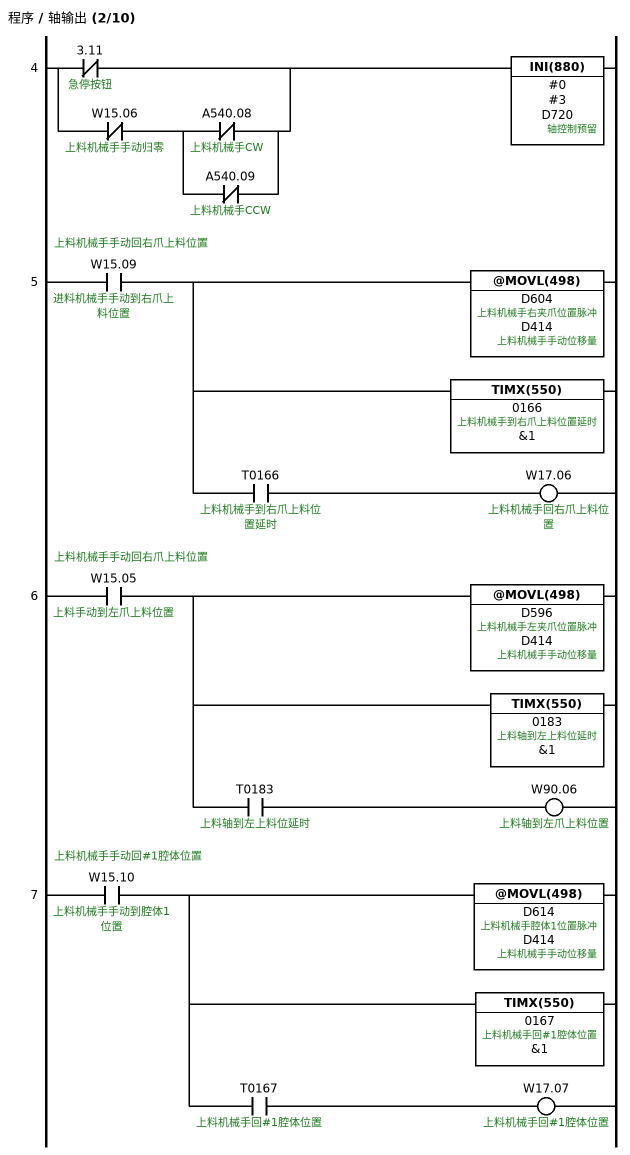
; [picture p144: 程序 / 轴输出, rungs 4-7]
; rung 4
LDNOT 3.11  ; 急停按钮
LDNOT W15.06  ; 上料机械手手动归零
LDNOT A540.08  ; 上料机械手CW
ORNOT A540.09  ; 上料机械手CCW
ANDLD
ORLD
INI(880) #0 #3 D720  ; 轴控制预留
; rung 5: 上料机械手手动回右爪上料位置
LD W15.09  ; 进料机械手手动到右爪上料位置
@MOVL(498) D604 D414  ; 上料机械手右夹爪位置脉冲, 上料机械手手动位移量
TIMX(550) 0166 &1  ; 上料机械手到右爪上料位置延时
AND T0166  ; 上料机械手到右爪上料位置延时
OUT W17.06  ; 上料机械手回右爪上料位置
; rung 6: 上料机械手手动回右爪上料位置
LD W15.05  ; 上料手动到左爪上料位置
@MOVL(498) D596 D414  ; 上料机械手左夹爪位置脉冲, 上料机械手手动位移量
TIMX(550) 0183 &1  ; 上料轴到左上料位延时
AND T0183  ; 上料轴到左上料位延时
OUT W90.06  ; 上料轴到左爪上料位置
; rung 7: 上料机械手手动回#1腔体位置
LD W15.10  ; 上料机械手手动到腔体1位置
@MOVL(498) D614 D414  ; 上料机械手腔体1位置脉冲, 上料机械手手动位移量
TIMX(550) 0167 &1  ; 上料机械手回#1腔体位置
AND T0167  ; 上料机械手回#1腔体位置
OUT W17.07  ; 上料机械手回#1腔体位置

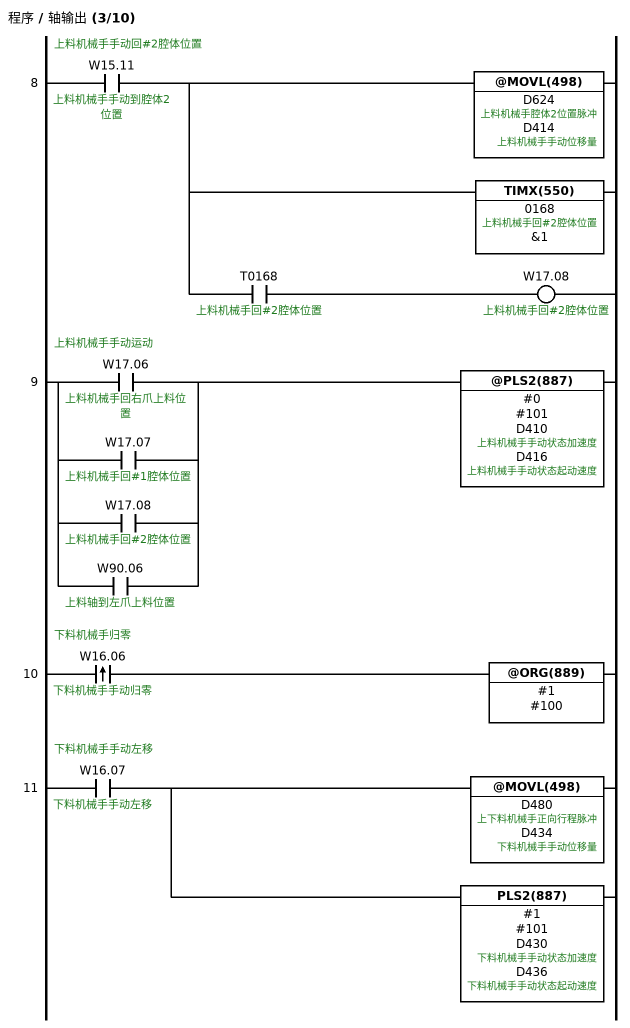
; rung 8: 上料机械手手动回#2腔体位置
LD W15.11  ; 上料机械手手动到腔体2位置
@MOVL(498) D624 D414  ; 上料机械手腔体2位置脉冲, 上料机械手手动位移量
TIMX(550) 0168 &1  ; 上料机械手回#2腔体位置
AND T0168  ; 上料机械手回#2腔体位置
OUT W17.08  ; 上料机械手回#2腔体位置
; rung 9: 上料机械手手动运动
LD W17.06  ; 上料机械手回右爪上料位置
OR W17.07  ; 上料机械手回#1腔体位置
OR W17.08  ; 上料机械手回#2腔体位置
OR W90.06  ; 上料轴到左爪上料位置
@PLS2(887) #0 #101 D410 D416  ; 上料机械手手动状态加速度, 上料机械手手动状态起动速度
; rung 10: 下料机械手归零
@LD W16.06  ; 下料机械手手动归零
@ORG(889) #1 #100
; rung 11: 下料机械手手动左移
LD W16.07  ; 下料机械手手动左移
@MOVL(498) D480 D434  ; 上下料机械手正向行程脉冲, 下料机械手手动位移量
PLS2(887) #1 #101 D430 D436  ; 下料机械手手动状态加速度, 下料机械手手动状态起动速度

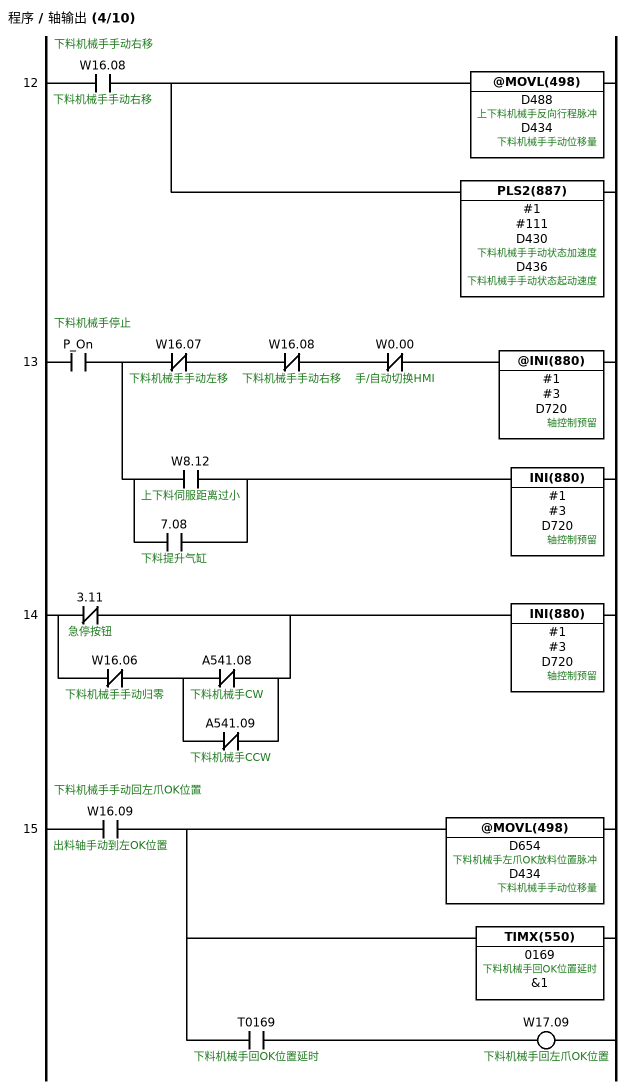
; rung 12: 下料机械手手动右移
LD W16.08  ; 下料机械手手动右移
@MOVL(498) D488 D434  ; 上下料机械手反向行程脉冲, 下料机械手手动位移量
PLS2(887) #1 #111 D430 D436  ; 下料机械手手动状态加速度, 下料机械手手动状态起动速度
; rung 13: 下料机械手停止
LD P_On
OUT TR0
ANDNOT W16.07  ; 下料机械手手动左移
ANDNOT W16.08  ; 下料机械手手动右移
ANDNOT W0.00  ; 手/自动切换HMI
@INI(880) #1 #3 D720  ; 轴控制预留
LD TR0
LD W8.12  ; 上下料伺服距离过小
OR 7.08  ; 下料提升气缸
ANDLD
INI(880) #1 #3 D720  ; 轴控制预留
; rung 14
LDNOT 3.11  ; 急停按钮
LDNOT W16.06  ; 下料机械手手动归零
LDNOT A541.08  ; 下料机械手CW
ORNOT A541.09  ; 下料机械手CCW
ANDLD
ORLD
INI(880) #1 #3 D720  ; 轴控制预留
; rung 15: 下料机械手手动回左爪OK位置
LD W16.09  ; 出料轴手动到左OK位置
@MOVL(498) D654 D434  ; 下料机械手左爪OK放料位置脉冲, 下料机械手手动位移量
TIMX(550) 0169 &1  ; 下料机械手回OK位置延时
AND T0169  ; 下料机械手回OK位置延时
OUT W17.09  ; 下料机械手回左爪OK位置

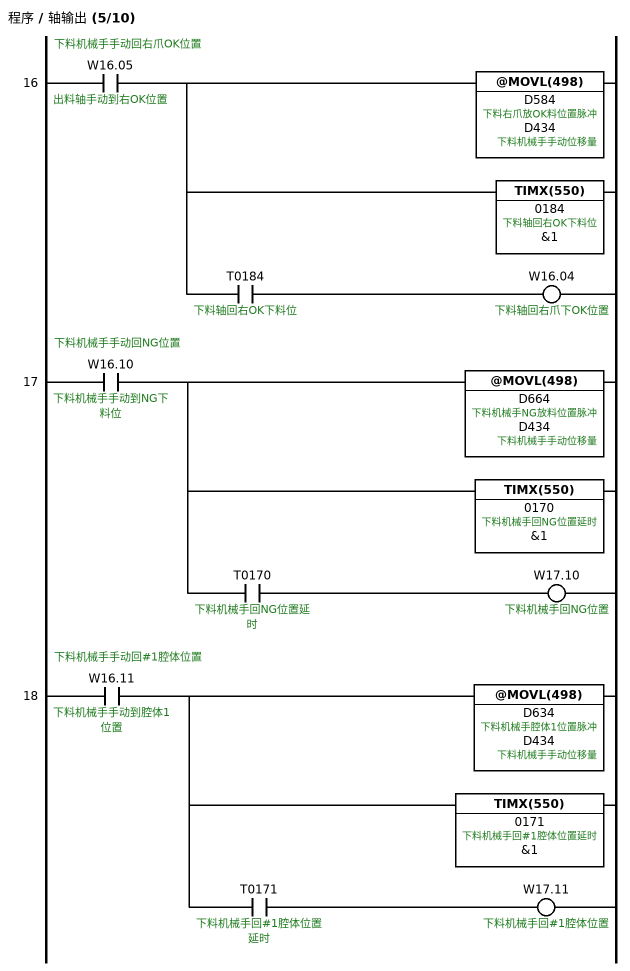
; rung 16: 下料机械手手动回右爪OK位置
LD W16.05  ; 出料轴手动到右OK位置
@MOVL(498) D584 D434  ; 下料右爪放OK料位置脉冲, 下料机械手手动位移量
TIMX(550) 0184 &1  ; 下料轴回右OK下料位
AND T0184  ; 下料轴回右OK下料位
OUT W16.04  ; 下料轴回右爪下OK位置
; rung 17: 下料机械手手动回NG位置
LD W16.10  ; 下料机械手手动到NG下料位
@MOVL(498) D664 D434  ; 下料机械手NG放料位置脉冲, 下料机械手手动位移量
TIMX(550) 0170 &1  ; 下料机械手回NG位置延时
AND T0170  ; 下料机械手回NG位置延时
OUT W17.10  ; 下料机械手回NG位置
; rung 18: 下料机械手手动回#1腔体位置
LD W16.11  ; 下料机械手手动到腔体1位置
@MOVL(498) D634 D434  ; 下料机械手腔体1位置脉冲, 下料机械手手动位移量
TIMX(550) 0171 &1  ; 下料机械手回#1腔体位置延时
AND T0171  ; 下料机械手回#1腔体位置延时
OUT W17.11  ; 下料机械手回#1腔体位置

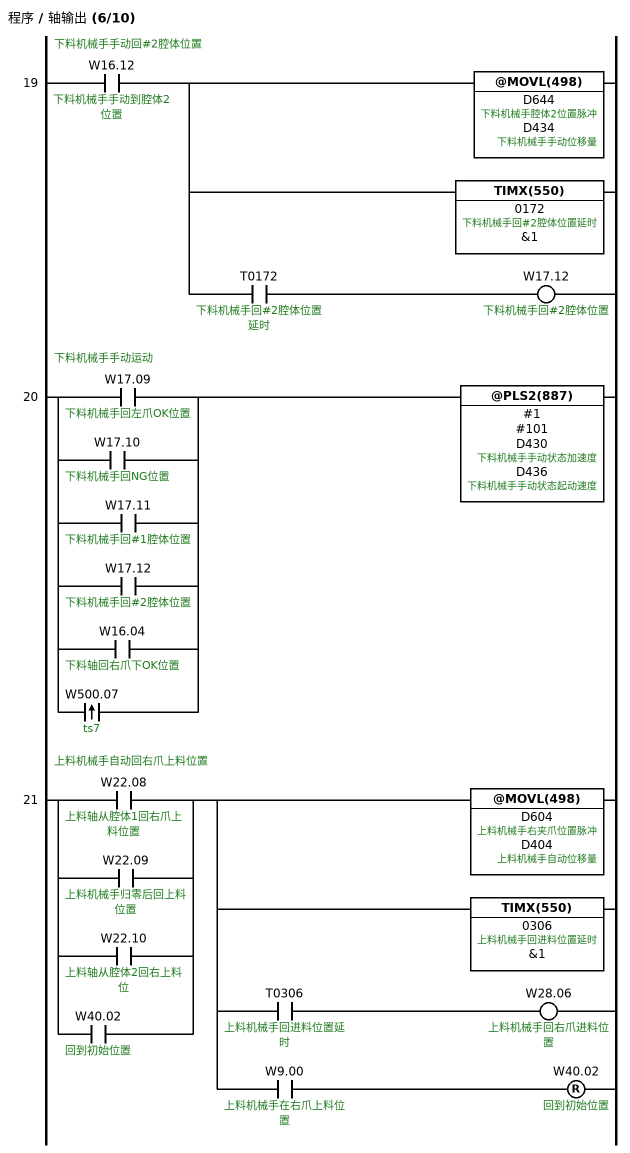
; rung 19: 下料机械手手动回#2腔体位置
LD W16.12  ; 下料机械手手动到腔体2位置
@MOVL(498) D644 D434  ; 下料机械手腔体2位置脉冲, 下料机械手手动位移量
TIMX(550) 0172 &1  ; 下料机械手回#2腔体位置延时
AND T0172  ; 下料机械手回#2腔体位置延时
OUT W17.12  ; 下料机械手回#2腔体位置
; rung 20: 下料机械手手动运动
LD W17.09  ; 下料机械手回左爪OK位置
OR W17.10  ; 下料机械手回NG位置
OR W17.11  ; 下料机械手回#1腔体位置
OR W17.12  ; 下料机械手回#2腔体位置
OR W16.04  ; 下料轴回右爪下OK位置
@OR W500.07  ; ts7
@PLS2(887) #1 #101 D430 D436  ; 下料机械手手动状态加速度, 下料机械手手动状态起动速度
; rung 21: 上料机械手自动回右爪上料位置
LD W22.08  ; 上料轴从腔体1回右爪上料位置
OR W22.09  ; 上料机械手归零后回上料位置
OR W22.10  ; 上料轴从腔体2回右上料位
OR W40.02  ; 回到初始位置
OUT TR0
@MOVL(498) D604 D404  ; 上料机械手右夹爪位置脉冲, 上料机械手自动位移量
TIMX(550) 0306 &1  ; 上料机械手回进料位置延时
AND T0306  ; 上料机械手回进料位置延时
OUT W28.06  ; 上料机械手回右爪进料位置
LD TR0
AND W9.00  ; 上料机械手在右爪上料位置
RSET W40.02  ; 回到初始位置

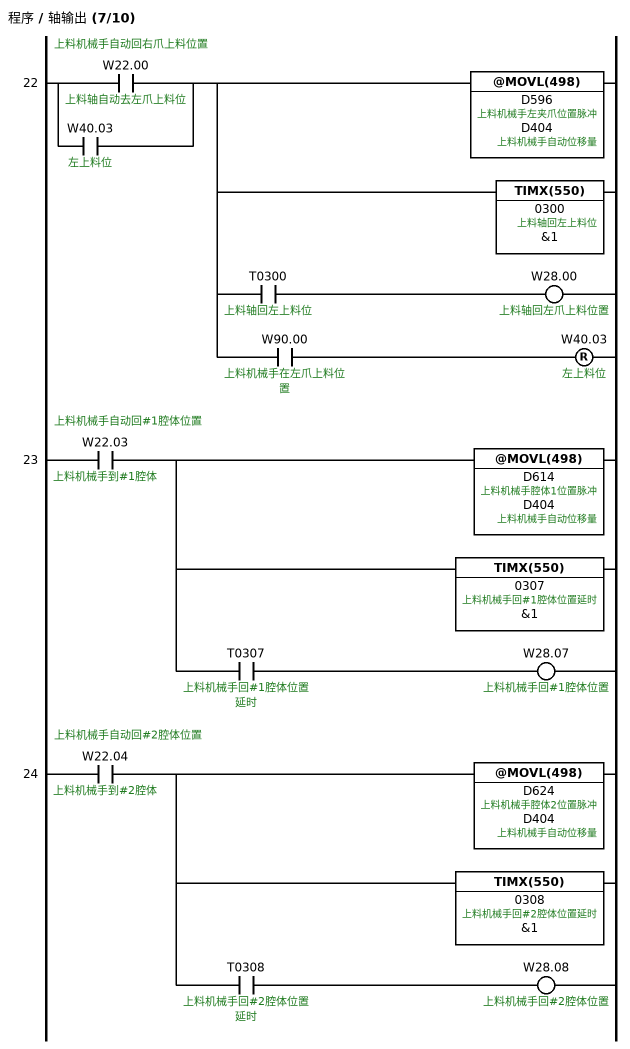
; rung 22: 上料机械手自动回右爪上料位置
LD W22.00  ; 上料轴自动去左爪上料位
OR W40.03  ; 左上料位
OUT TR0
@MOVL(498) D596 D404  ; 上料机械手左夹爪位置脉冲, 上料机械手自动位移量
TIMX(550) 0300 &1  ; 上料轴回左上料位
AND T0300  ; 上料轴回左上料位
OUT W28.00  ; 上料轴回左爪上料位置
LD TR0
AND W90.00  ; 上料机械手在左爪上料位置
RSET W40.03  ; 左上料位
; rung 23: 上料机械手自动回#1腔体位置
LD W22.03  ; 上料机械手到#1腔体
@MOVL(498) D614 D404  ; 上料机械手腔体1位置脉冲, 上料机械手自动位移量
TIMX(550) 0307 &1  ; 上料机械手回#1腔体位置延时
AND T0307  ; 上料机械手回#1腔体位置延时
OUT W28.07  ; 上料机械手回#1腔体位置
; rung 24: 上料机械手自动回#2腔体位置
LD W22.04  ; 上料机械手到#2腔体
@MOVL(498) D624 D404  ; 上料机械手腔体2位置脉冲, 上料机械手自动位移量
TIMX(550) 0308 &1  ; 上料机械手回#2腔体位置延时
AND T0308  ; 上料机械手回#2腔体位置延时
OUT W28.08  ; 上料机械手回#2腔体位置

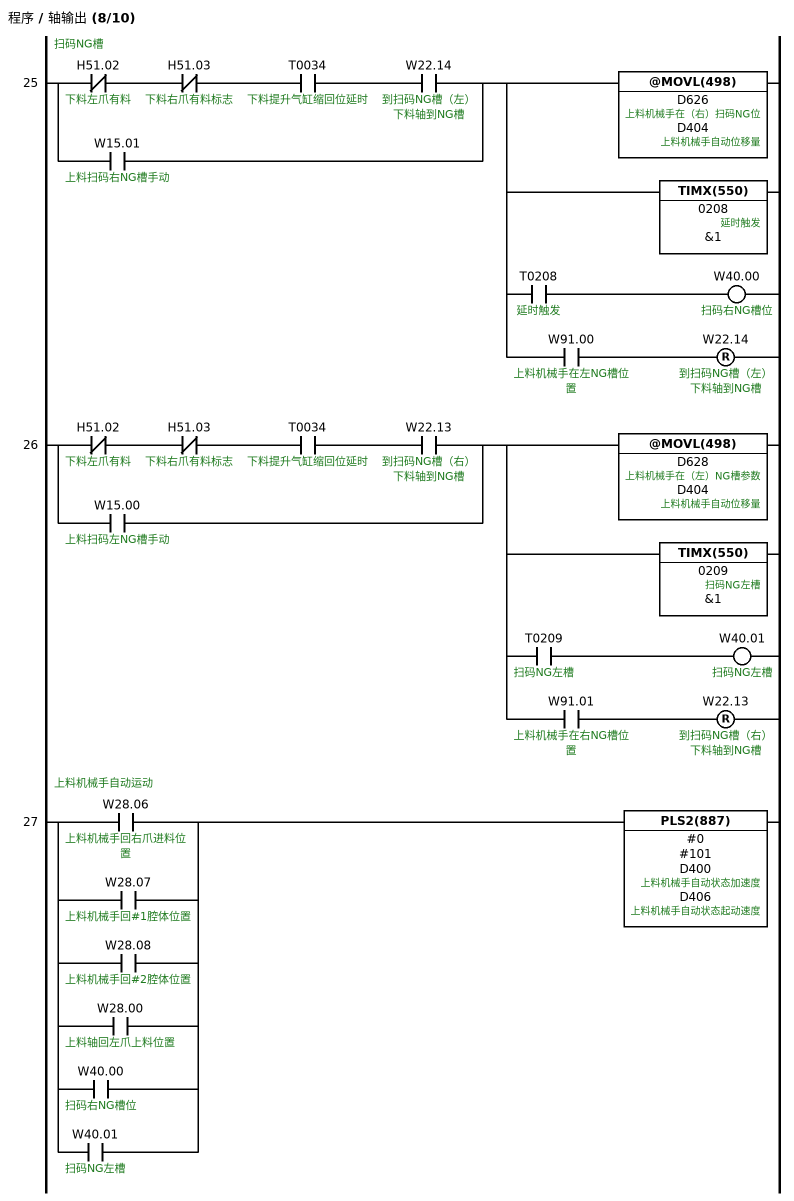
; rung 25: 扫码NG槽
LDNOT H51.02  ; 下料左爪有料
ANDNOT H51.03  ; 下料右爪有料标志
AND T0034  ; 下料提升气缸缩回位延时
AND W22.14  ; 到扫码NG槽（左） 下料轴到NG槽
OR W15.01  ; 上料扫码右NG槽手动
OUT TR0
@MOVL(498) D626 D404  ; 上料机械手在（右）扫码NG位, 上料机械手自动位移量
TIMX(550) 0208 &1  ; 延时触发
AND T0208  ; 延时触发
OUT W40.00  ; 扫码右NG槽位
LD TR0
AND W91.00  ; 上料机械手在左NG槽位置
RSET W22.14  ; 到扫码NG槽（左） 下料轴到NG槽
; rung 26
LDNOT H51.02  ; 下料左爪有料
ANDNOT H51.03  ; 下料右爪有料标志
AND T0034  ; 下料提升气缸缩回位延时
AND W22.13  ; 到扫码NG槽（右） 下料轴到NG槽
OR W15.00  ; 上料扫码左NG槽手动
OUT TR0
@MOVL(498) D628 D404  ; 上料机械手在（左）NG槽参数, 上料机械手自动位移量
TIMX(550) 0209 &1  ; 扫码NG左槽
AND T0209  ; 扫码NG左槽
OUT W40.01  ; 扫码NG左槽
LD TR0
AND W91.01  ; 上料机械手在右NG槽位置
RSET W22.13  ; 到扫码NG槽（右） 下料轴到NG槽
; rung 27: 上料机械手自动运动
LD W28.06  ; 上料机械手回右爪进料位置
OR W28.07  ; 上料机械手回#1腔体位置
OR W28.08  ; 上料机械手回#2腔体位置
OR W28.00  ; 上料轴回左爪上料位置
OR W40.00  ; 扫码右NG槽位
OR W40.01  ; 扫码NG左槽
PLS2(887) #0 #101 D400 D406  ; 上料机械手自动状态加速度, 上料机械手自动状态起动速度

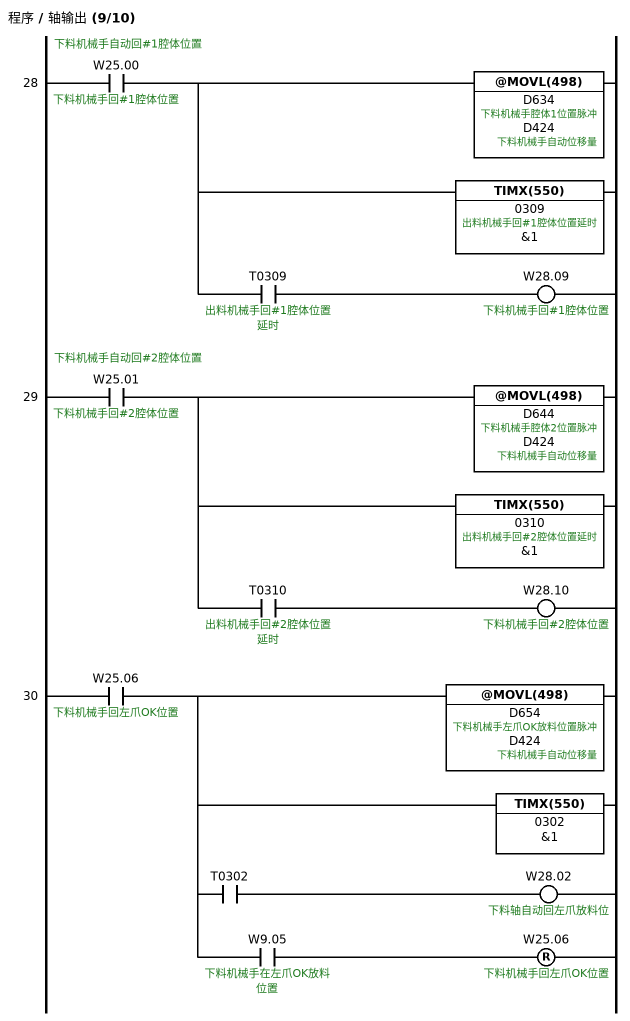
; rung 28: 下料机械手自动回#1腔体位置
LD W25.00  ; 下料机械手回#1腔体位置
@MOVL(498) D634 D424  ; 下料机械手腔体1位置脉冲, 下料机械手自动位移量
TIMX(550) 0309 &1  ; 出料机械手回#1腔体位置延时
AND T0309  ; 出料机械手回#1腔体位置延时
OUT W28.09  ; 下料机械手回#1腔体位置
; rung 29: 下料机械手自动回#2腔体位置
LD W25.01  ; 下料机械手回#2腔体位置
@MOVL(498) D644 D424  ; 下料机械手腔体2位置脉冲, 下料机械手自动位移量
TIMX(550) 0310 &1  ; 出料机械手回#2腔体位置延时
AND T0310  ; 出料机械手回#2腔体位置延时
OUT W28.10  ; 下料机械手回#2腔体位置
; rung 30
LD W25.06  ; 下料机械手回左爪OK位置
OUT TR0
@MOVL(498) D654 D424  ; 下料机械手左爪OK放料位置脉冲, 下料机械手自动位移量
TIMX(550) 0302 &1
AND T0302
OUT W28.02  ; 下料轴自动回左爪放料位
LD TR0
AND W9.05  ; 下料机械手在左爪OK放料位置
RSET W25.06  ; 下料机械手回左爪OK位置

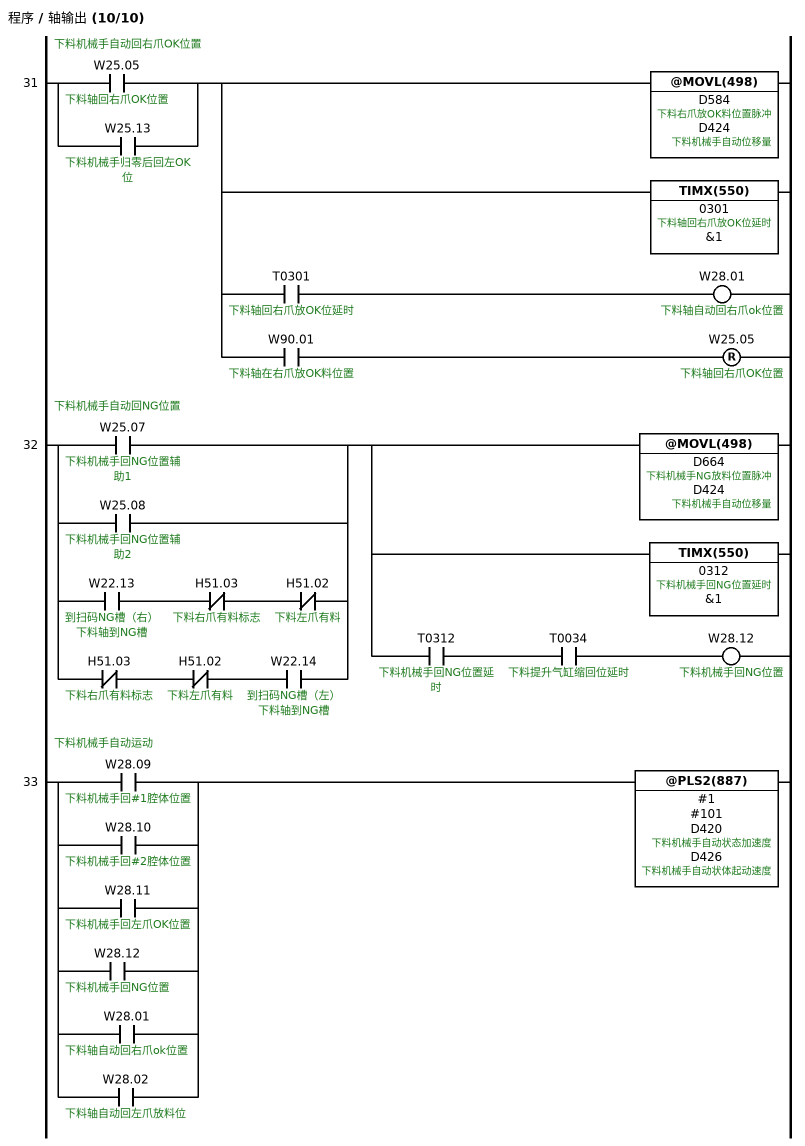
; rung 31: 下料机械手自动回右爪OK位置
LD W25.05  ; 下料轴回右爪OK位置
OR W25.13  ; 下料机械手归零后回左OK位
OUT TR0
@MOVL(498) D584 D424  ; 下料右爪放OK料位置脉冲, 下料机械手自动位移量
TIMX(550) 0301 &1  ; 下料轴回右爪放OK位延时
AND T0301  ; 下料轴回右爪放OK位延时
OUT W28.01  ; 下料轴自动回右爪ok位置
LD TR0
AND W90.01  ; 下料轴在右爪放OK料位置
RSET W25.05  ; 下料轴回右爪OK位置
; rung 32: 下料机械手自动回NG位置
LD W25.07  ; 下料机械手回NG位置辅助1
OR W25.08  ; 下料机械手回NG位置辅助2
LD W22.13  ; 到扫码NG槽（右） 下料轴到NG槽
ANDNOT H51.03  ; 下料右爪有料标志
ANDNOT H51.02  ; 下料左爪有料
ORLD
LDNOT H51.03  ; 下料右爪有料标志
ANDNOT H51.02  ; 下料左爪有料
AND W22.14  ; 到扫码NG槽（左） 下料轴到NG槽
ORLD
@MOVL(498) D664 D424  ; 下料机械手NG放料位置脉冲, 下料机械手自动位移量
TIMX(550) 0312 &1  ; 下料机械手回NG位置延时
AND T0312  ; 下料机械手回NG位置延时
AND T0034  ; 下料提升气缸缩回位延时
OUT W28.12  ; 下料机械手回NG位置
; rung 33: 下料机械手自动运动
LD W28.09  ; 下料机械手回#1腔体位置
OR W28.10  ; 下料机械手回#2腔体位置
OR W28.11  ; 下料机械手回左爪OK位置
OR W28.12  ; 下料机械手回NG位置
OR W28.01  ; 下料轴自动回右爪ok位置
OR W28.02  ; 下料轴自动回左爪放料位
@PLS2(887) #1 #101 D420 D426  ; 下料机械手自动状态加速度, 下料机械手自动状体起动速度

### Section 普通输出

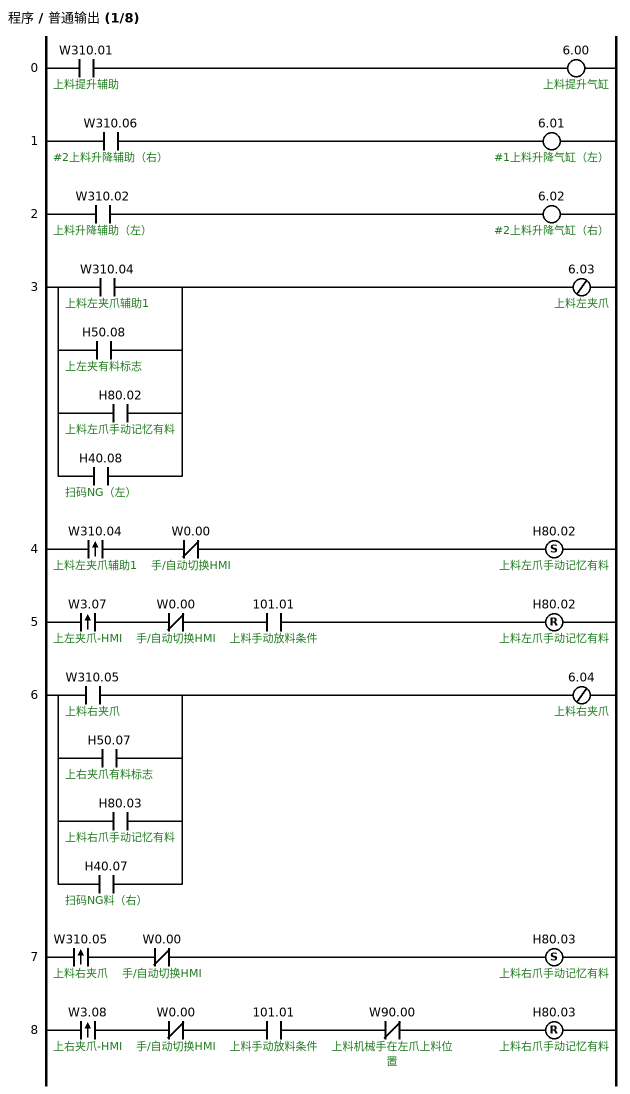
; rung 0
LD W310.01  ; 上料提升辅助
OUT 6.00  ; 上料提升气缸
; rung 1
LD W310.06  ; #2上料升降辅助（右）
OUT 6.01  ; #1上料升降气缸（左）
; rung 2
LD W310.02  ; 上料升降辅助（左）
OUT 6.02  ; #2上料升降气缸（右）
; rung 3
LD W310.04  ; 上料左夹爪辅助1
OR H50.08  ; 上左夹有料标志
OR H80.02  ; 上料左爪手动记忆有料
OR H40.08  ; 扫码NG（左）
OUTNOT 6.03  ; 上料左夹爪
; rung 4
@LD W310.04  ; 上料左夹爪辅助1
ANDNOT W0.00  ; 手/自动切换HMI
SET H80.02  ; 上料左爪手动记忆有料
; rung 5
@LD W3.07  ; 上左夹爪-HMI
ANDNOT W0.00  ; 手/自动切换HMI
AND 101.01  ; 上料手动放料条件
RSET H80.02  ; 上料左爪手动记忆有料
; rung 6
LD W310.05  ; 上料右夹爪
OR H50.07  ; 上右夹爪有料标志
OR H80.03  ; 上料右爪手动记忆有料
OR H40.07  ; 扫码NG料（右）
OUTNOT 6.04  ; 上料右夹爪
; rung 7
@LD W310.05  ; 上料右夹爪
ANDNOT W0.00  ; 手/自动切换HMI
SET H80.03  ; 上料右爪手动记忆有料
; rung 8
@LD W3.08  ; 上右夹爪-HMI
ANDNOT W0.00  ; 手/自动切换HMI
AND 101.01  ; 上料手动放料条件
ANDNOT W90.00  ; 上料机械手在左爪上料位置
RSET H80.03  ; 上料右爪手动记忆有料

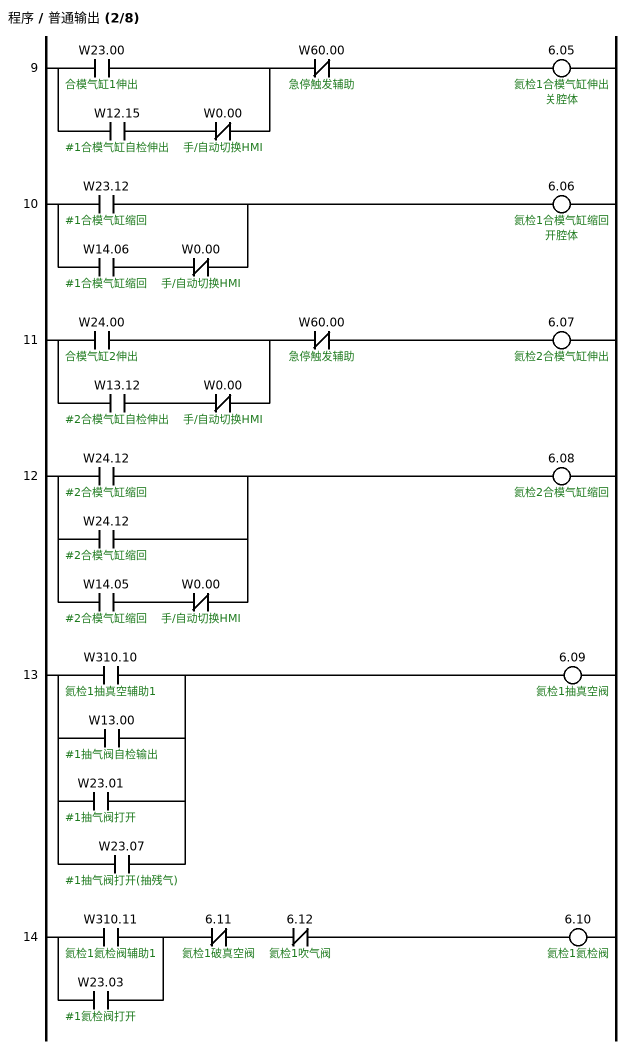
; rung 9
LD W23.00  ; 合模气缸1伸出
LD W12.15  ; #1合模气缸自检伸出
ANDNOT W0.00  ; 手/自动切换HMI
ORLD
ANDNOT W60.00  ; 急停触发辅助
OUT 6.05  ; 氦检1合模气缸伸出 关腔体
; rung 10
LD W23.12  ; #1合模气缸缩回
LD W14.06  ; #1合模气缸缩回
ANDNOT W0.00  ; 手/自动切换HMI
ORLD
OUT 6.06  ; 氦检1合模气缸缩回 开腔体
; rung 11
LD W24.00  ; 合模气缸2伸出
LD W13.12  ; #2合模气缸自检伸出
ANDNOT W0.00  ; 手/自动切换HMI
ORLD
ANDNOT W60.00  ; 急停触发辅助
OUT 6.07  ; 氦检2合模气缸伸出
; rung 12
LD W24.12  ; #2合模气缸缩回
OR W24.12  ; #2合模气缸缩回
LD W14.05  ; #2合模气缸缩回
ANDNOT W0.00  ; 手/自动切换HMI
ORLD
OUT 6.08  ; 氦检2合模气缸缩回
; rung 13
LD W310.10  ; 氦检1抽真空辅助1
OR W13.00  ; #1抽气阀自检输出
OR W23.01  ; #1抽气阀打开
OR W23.07  ; #1抽气阀打开(抽残气)
OUT 6.09  ; 氦检1抽真空阀
; rung 14
LD W310.11  ; 氦检1氦检阀辅助1
OR W23.03  ; #1氦检阀打开
ANDNOT 6.11  ; 氦检1破真空阀
ANDNOT 6.12  ; 氦检1吹气阀
OUT 6.10  ; 氦检1氦检阀

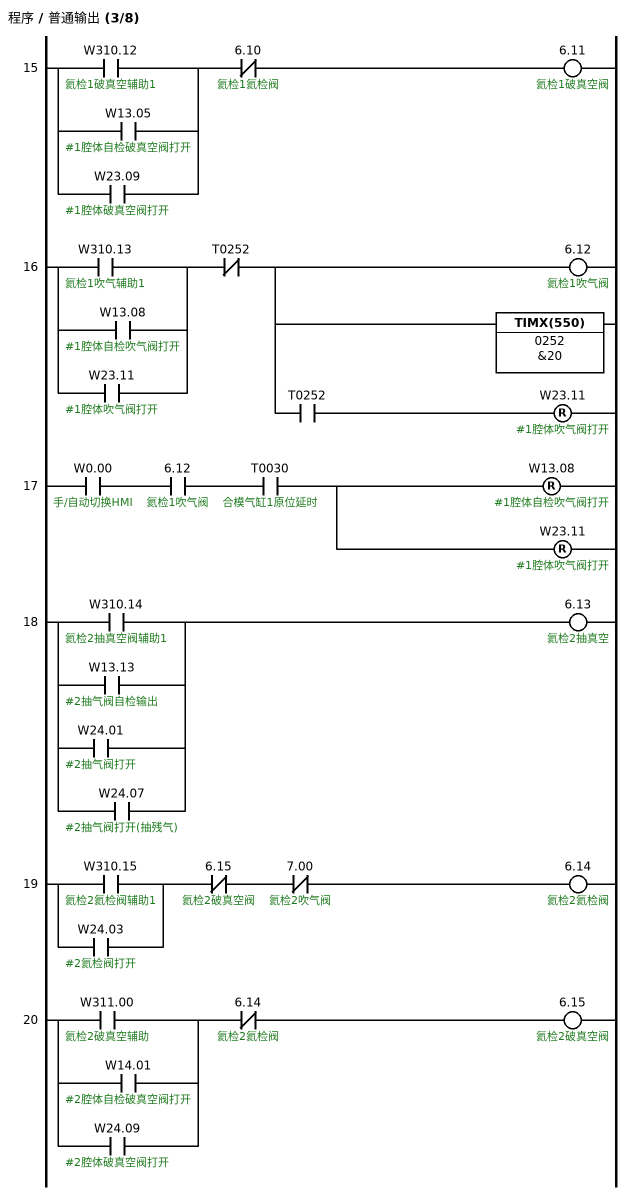
; rung 15
LD W310.12  ; 氦检1破真空辅助1
OR W13.05  ; #1腔体自检破真空阀打开
OR W23.09  ; #1腔体破真空阀打开
ANDNOT 6.10  ; 氦检1氦检阀
OUT 6.11  ; 氦检1破真空阀
; rung 16
LD W310.13  ; 氦检1吹气辅助1
OR W13.08  ; #1腔体自检吹气阀打开
OR W23.11  ; #1腔体吹气阀打开
ANDNOT T0252
OUT 6.12  ; 氦检1吹气阀
TIMX(550) 0252 &20
AND T0252
RSET W23.11  ; #1腔体吹气阀打开
; rung 17
LD W0.00  ; 手/自动切换HMI
AND 6.12  ; 氦检1吹气阀
AND T0030  ; 合模气缸1原位延时
RSET W13.08  ; #1腔体自检吹气阀打开
RSET W23.11  ; #1腔体吹气阀打开
; rung 18
LD W310.14  ; 氦检2抽真空阀辅助1
OR W13.13  ; #2抽气阀自检输出
OR W24.01  ; #2抽气阀打开
OR W24.07  ; #2抽气阀打开(抽残气)
OUT 6.13  ; 氦检2抽真空
; rung 19
LD W310.15  ; 氦检2氦检阀辅助1
OR W24.03  ; #2氦检阀打开
ANDNOT 6.15  ; 氦检2破真空阀
ANDNOT 7.00  ; 氦检2吹气阀
OUT 6.14  ; 氦检2氦检阀
; rung 20
LD W311.00  ; 氦检2破真空辅助
OR W14.01  ; #2腔体自检破真空阀打开
OR W24.09  ; #2腔体破真空阀打开
ANDNOT 6.14  ; 氦检2氦检阀
OUT 6.15  ; 氦检2破真空阀

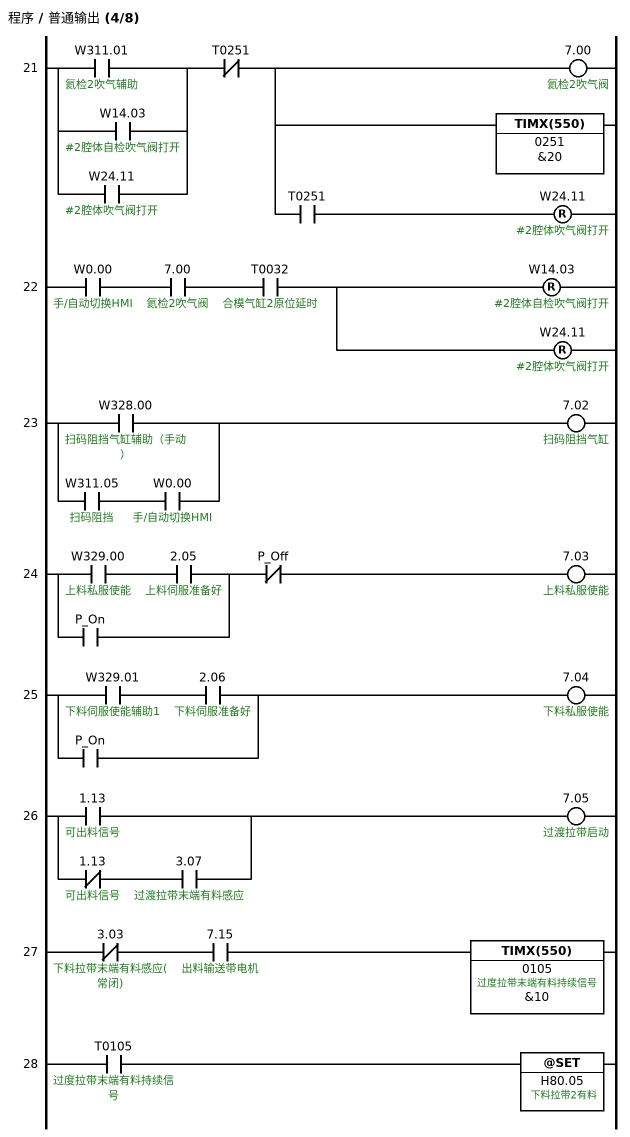
; rung 21
LD W311.01  ; 氦检2吹气辅助
OR W14.03  ; #2腔体自检吹气阀打开
OR W24.11  ; #2腔体吹气阀打开
ANDNOT T0251
OUT 7.00  ; 氦检2吹气阀
TIMX(550) 0251 &20
AND T0251
RSET W24.11  ; #2腔体吹气阀打开
; rung 22
LD W0.00  ; 手/自动切换HMI
AND 7.00  ; 氦检2吹气阀
AND T0032  ; 合模气缸2原位延时
RSET W14.03  ; #2腔体自检吹气阀打开
RSET W24.11  ; #2腔体吹气阀打开
; rung 23
LD W328.00  ; 扫码阻挡气缸辅助（手动）
LD W311.05  ; 扫码阻挡
AND W0.00  ; 手/自动切换HMI
ORLD
OUT 7.02  ; 扫码阻挡气缸
; rung 24
LD W329.00  ; 上料私服使能
AND 2.05  ; 上料伺服准备好
OR P_On
ANDNOT P_Off
OUT 7.03  ; 上料私服使能
; rung 25
LD W329.01  ; 下料伺服使能辅助1
AND 2.06  ; 下料伺服准备好
OR P_On
OUT 7.04  ; 下料私服使能
; rung 26
LD 1.13  ; 可出料信号
LDNOT 1.13  ; 可出料信号
AND 3.07  ; 过渡拉带末端有料感应
ORLD
OUT 7.05  ; 过渡拉带启动
; rung 27
LDNOT 3.03  ; 下料拉带末端有料感应(常闭)
AND 7.15  ; 出料输送带电机
TIMX(550) 0105 &10  ; 过度拉带末端有料持续信号
; rung 28
LD T0105  ; 过度拉带末端有料持续信号
@SET H80.05  ; 下料拉带2有料

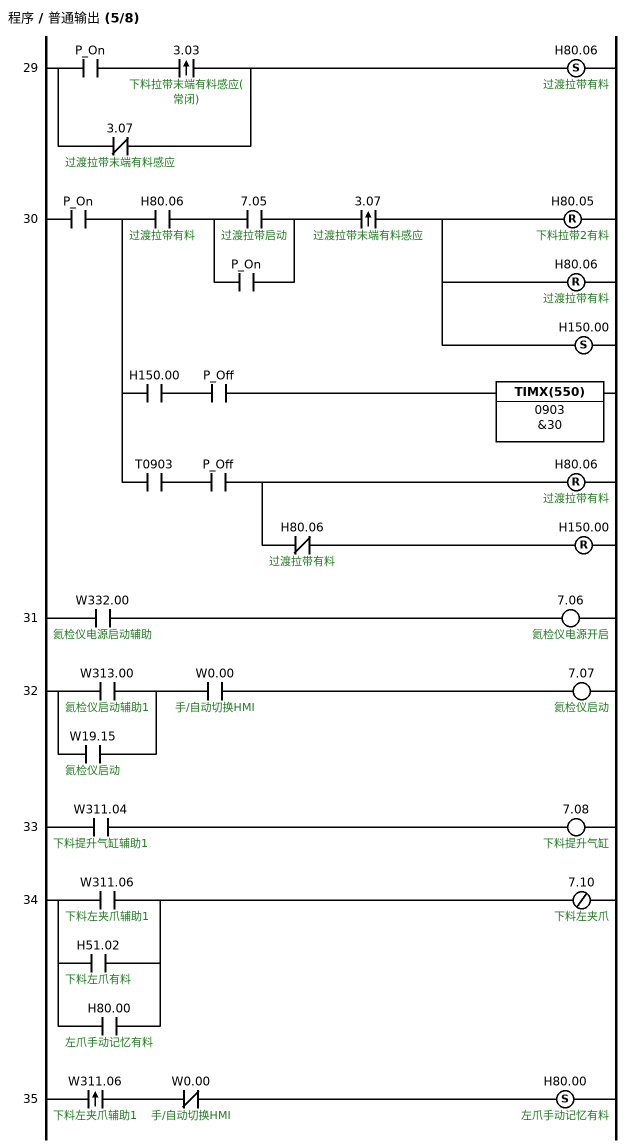
; rung 29
LD P_On
@AND 3.03  ; 下料拉带末端有料感应(常闭)
ORNOT 3.07  ; 过渡拉带末端有料感应
SET H80.06  ; 过渡拉带有料
; rung 30
LD P_On
OUT TR0
AND H80.06  ; 过渡拉带有料
LD 7.05  ; 过渡拉带启动
OR P_On
ANDLD
@AND 3.07  ; 过渡拉带末端有料感应
RSET H80.05  ; 下料拉带2有料
RSET H80.06  ; 过渡拉带有料
SET H150.00
LD TR0
AND H150.00
AND P_Off
TIMX(550) 0903 &30
LD TR0
AND T0903
AND P_Off
RSET H80.06  ; 过渡拉带有料
ANDNOT H80.06  ; 过渡拉带有料
RSET H150.00
; rung 31
LD W332.00  ; 氦检仪电源启动辅助
OUT 7.06  ; 氦检仪电源开启
; rung 32
LD W313.00  ; 氦检仪启动辅助1
OR W19.15  ; 氦检仪启动
AND W0.00  ; 手/自动切换HMI
OUT 7.07  ; 氦检仪启动
; rung 33
LD W311.04  ; 下料提升气缸辅助1
OUT 7.08  ; 下料提升气缸
; rung 34
LD W311.06  ; 下料左夹爪辅助1
OR H51.02  ; 下料左爪有料
OR H80.00  ; 左爪手动记忆有料
OUTNOT 7.10  ; 下料左夹爪
; rung 35
@LD W311.06  ; 下料左夹爪辅助1
ANDNOT W0.00  ; 手/自动切换HMI
SET H80.00  ; 左爪手动记忆有料

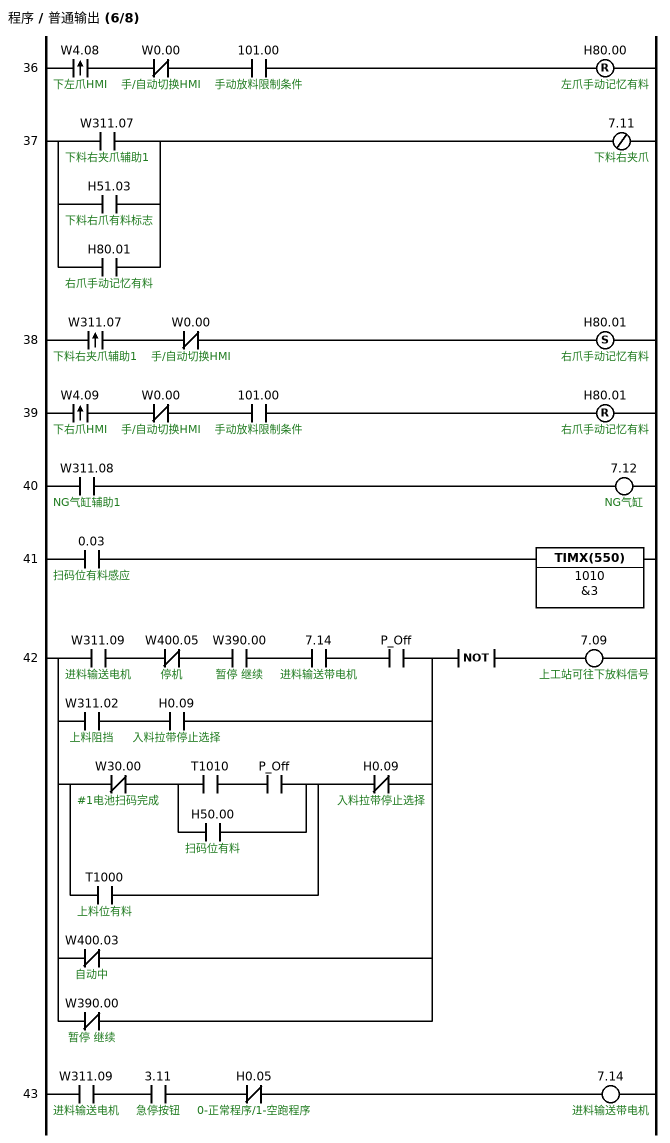
; rung 36
@LD W4.08  ; 下左爪HMI
ANDNOT W0.00  ; 手/自动切换HMI
AND 101.00  ; 手动放料限制条件
RSET H80.00  ; 左爪手动记忆有料
; rung 37
LD W311.07  ; 下料右夹爪辅助1
OR H51.03  ; 下料右爪有料标志
OR H80.01  ; 右爪手动记忆有料
OUTNOT 7.11  ; 下料右夹爪
; rung 38
@LD W311.07  ; 下料右夹爪辅助1
ANDNOT W0.00  ; 手/自动切换HMI
SET H80.01  ; 右爪手动记忆有料
; rung 39
@LD W4.09  ; 下右爪HMI
ANDNOT W0.00  ; 手/自动切换HMI
AND 101.00  ; 手动放料限制条件
RSET H80.01  ; 右爪手动记忆有料
; rung 40
LD W311.08  ; NG气缸辅助1
OUT 7.12  ; NG气缸
; rung 41
LD 0.03  ; 扫码位有料感应
TIMX(550) 1010 &3
; rung 42
LD W311.09  ; 进料输送电机
ANDNOT W400.05  ; 停机
AND W390.00  ; 暂停 继续
AND 7.14  ; 进料输送带电机
AND P_Off
LD W311.02  ; 上料阻挡
AND H0.09  ; 入料拉带停止选择
ORLD
LDNOT W30.00  ; #1电池扫码完成
LD T1010
AND P_Off
OR H50.00  ; 扫码位有料
ANDLD
OR T1000  ; 上料位有料
ANDNOT H0.09  ; 入料拉带停止选择
ORLD
ORNOT W400.03  ; 自动中
ORNOT W390.00  ; 暂停 继续
NOT(520)
OUT 7.09  ; 上工站可往下放料信号
; rung 43
LD W311.09  ; 进料输送电机
AND 3.11  ; 急停按钮
ANDNOT H0.05  ; 0-正常程序/1-空跑程序
OUT 7.14  ; 进料输送带电机

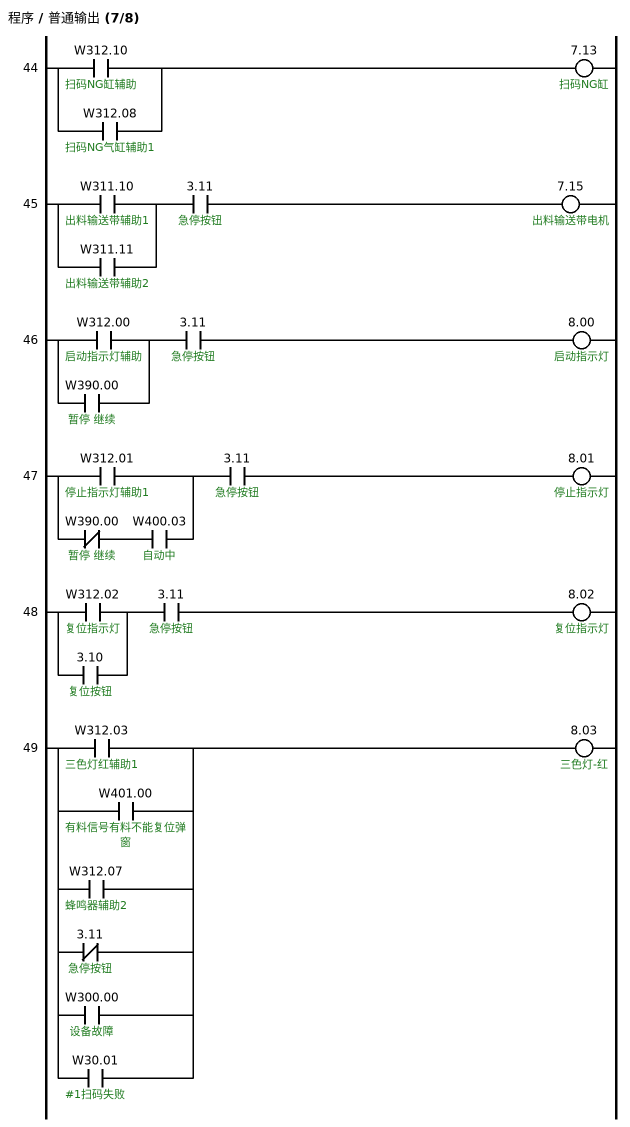
; rung 44
LD W312.10  ; 扫码NG缸辅助
OR W312.08  ; 扫码NG气缸辅助1
OUT 7.13  ; 扫码NG缸
; rung 45
LD W311.10  ; 出料输送带辅助1
OR W311.11  ; 出料输送带辅助2
AND 3.11  ; 急停按钮
OUT 7.15  ; 出料输送带电机
; rung 46
LD W312.00  ; 启动指示灯辅助
OR W390.00  ; 暂停 继续
AND 3.11  ; 急停按钮
OUT 8.00  ; 启动指示灯
; rung 47
LD W312.01  ; 停止指示灯辅助1
LDNOT W390.00  ; 暂停 继续
AND W400.03  ; 自动中
ORLD
AND 3.11  ; 急停按钮
OUT 8.01  ; 停止指示灯
; rung 48
LD W312.02  ; 复位指示灯
OR 3.10  ; 复位按钮
AND 3.11  ; 急停按钮
OUT 8.02  ; 复位指示灯
; rung 49
LD W312.03  ; 三色灯红辅助1
OR W401.00  ; 有料信号有料不能复位弹窗
OR W312.07  ; 蜂鸣器辅助2
ORNOT 3.11  ; 急停按钮
OR W300.00  ; 设备故障
OR W30.01  ; #1扫码失败
OUT 8.03  ; 三色灯-红

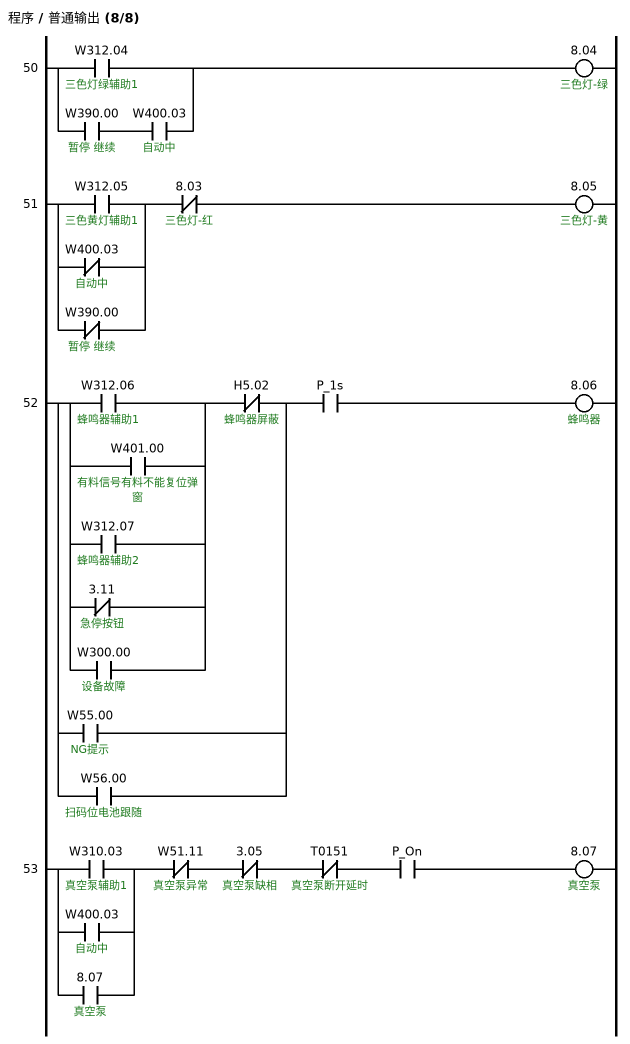
; rung 50
LD W312.04  ; 三色灯绿辅助1
LD W390.00  ; 暂停 继续
AND W400.03  ; 自动中
ORLD
OUT 8.04  ; 三色灯-绿
; rung 51
LD W312.05  ; 三色黄灯辅助1
ORNOT W400.03  ; 自动中
ORNOT W390.00  ; 暂停 继续
ANDNOT 8.03  ; 三色灯-红
OUT 8.05  ; 三色灯-黄
; rung 52
LD W312.06  ; 蜂鸣器辅助1
OR W401.00  ; 有料信号有料不能复位弹窗
OR W312.07  ; 蜂鸣器辅助2
ORNOT 3.11  ; 急停按钮
OR W300.00  ; 设备故障
ANDNOT H5.02  ; 蜂鸣器屏蔽
OR W55.00  ; NG提示
OR W56.00  ; 扫码位电池跟随
AND P_1s
OUT 8.06  ; 蜂鸣器
; rung 53
LD W310.03  ; 真空泵辅助1
OR W400.03  ; 自动中
OR 8.07  ; 真空泵
ANDNOT W51.11  ; 真空泵异常
ANDNOT 3.05  ; 真空泵缺相
ANDNOT T0151  ; 真空泵断开延时
AND P_On
OUT 8.07  ; 真空泵

### Section 氦检仪读值

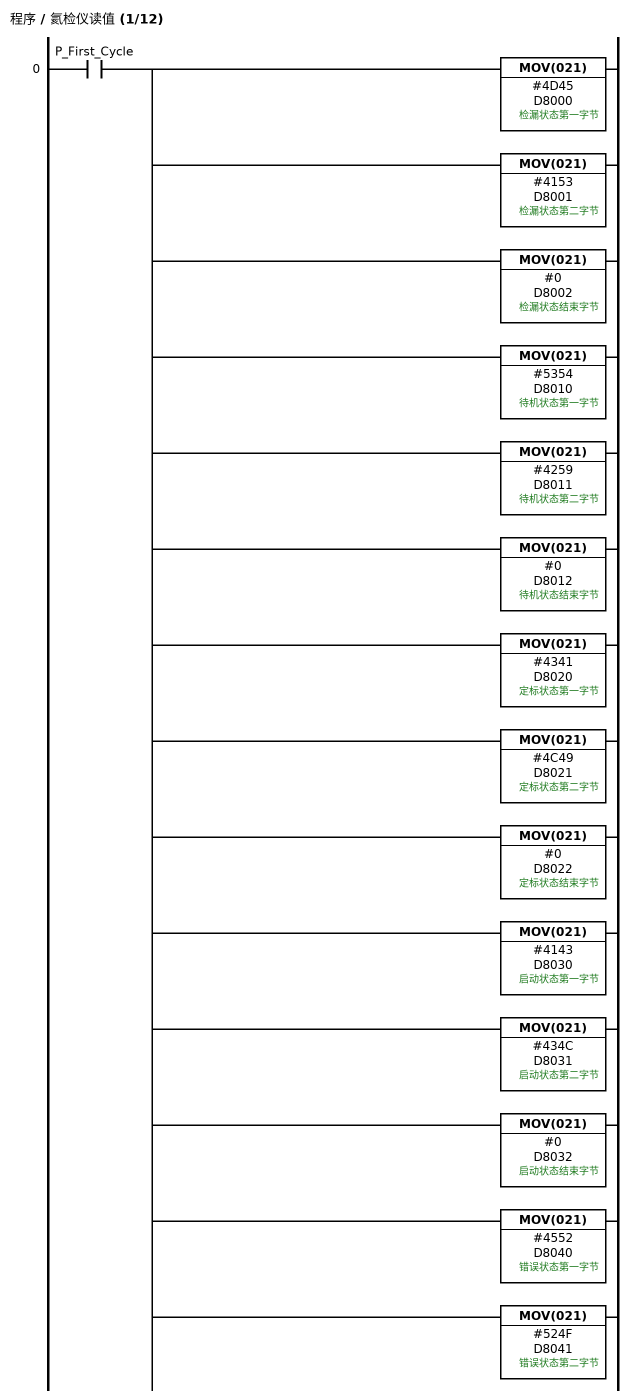

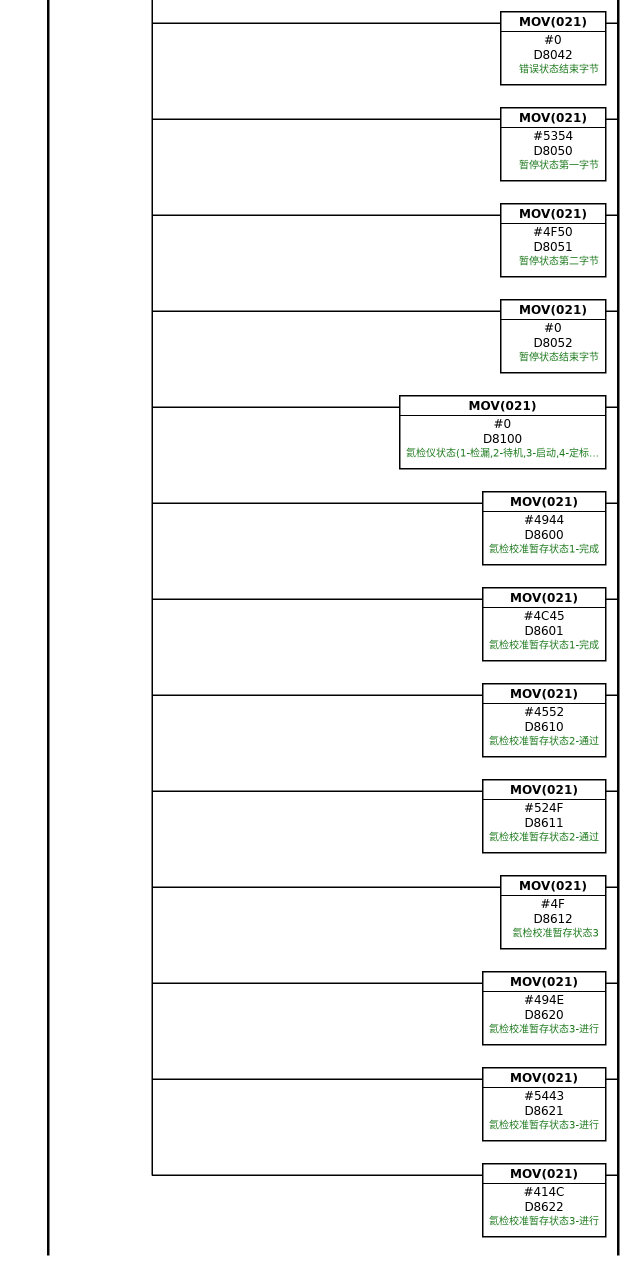
; rung 0
LD P_First_Cycle
MOV(021) #4D45 D8000  ; 检漏状态第一字节
MOV(021) #4153 D8001  ; 检漏状态第二字节
MOV(021) #0 D8002  ; 检漏状态结束字节
MOV(021) #5354 D8010  ; 待机状态第一字节
MOV(021) #4259 D8011  ; 待机状态第二字节
MOV(021) #0 D8012  ; 待机状态结束字节
MOV(021) #4341 D8020  ; 定标状态第一字节
MOV(021) #4C49 D8021  ; 定标状态第二字节
MOV(021) #0 D8022  ; 定标状态结束字节
MOV(021) #4143 D8030  ; 启动状态第一字节
MOV(021) #434C D8031  ; 启动状态第二字节
MOV(021) #0 D8032  ; 启动状态结束字节
MOV(021) #4552 D8040  ; 错误状态第一字节
MOV(021) #524F D8041  ; 错误状态第二字节
MOV(021) #0 D8042  ; 错误状态结束字节
MOV(021) #5354 D8050  ; 暂停状态第一字节
MOV(021) #4F50 D8051  ; 暂停状态第二字节
MOV(021) #0 D8052  ; 暂停状态结束字节
MOV(021) #0 D8100  ; 氦检仪状态(1-检漏,2-待机,3-启动,4-定标,5-错误,6-暂停)
MOV(021) #4944 D8600  ; 氦检校准暂存状态1-完成
MOV(021) #4C45 D8601  ; 氦检校准暂存状态1-完成
MOV(021) #4552 D8610  ; 氦检校准暂存状态2-通过
MOV(021) #524F D8611  ; 氦检校准暂存状态2-通过
MOV(021) #4F D8612  ; 氦检校准暂存状态3
MOV(021) #494E D8620  ; 氦检校准暂存状态3-进行
MOV(021) #5443 D8621  ; 氦检校准暂存状态3-进行
MOV(021) #414C D8622  ; 氦检校准暂存状态3-进行

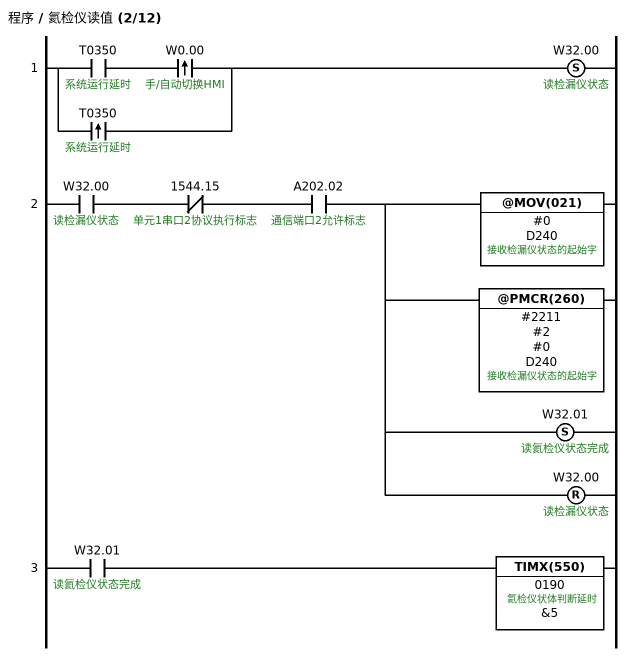
; rung 1
LD T0350  ; 系统运行延时
@AND W0.00  ; 手/自动切换HMI
@OR T0350  ; 系统运行延时
SET W32.00  ; 读检漏仪状态
; rung 2
LD W32.00  ; 读检漏仪状态
ANDNOT 1544.15  ; 单元1串口2协议执行标志
AND A202.02  ; 通信端口2允许标志
@MOV(021) #0 D240  ; 接收检漏仪状态的起始字
@PMCR(260) #2211 #2 #0 D240  ; 接收检漏仪状态的起始字
SET W32.01  ; 读氦检仪状态完成
RSET W32.00  ; 读检漏仪状态
; rung 3
LD W32.01  ; 读氦检仪状态完成
TIMX(550) 0190 &5  ; 氦检仪状体判断延时

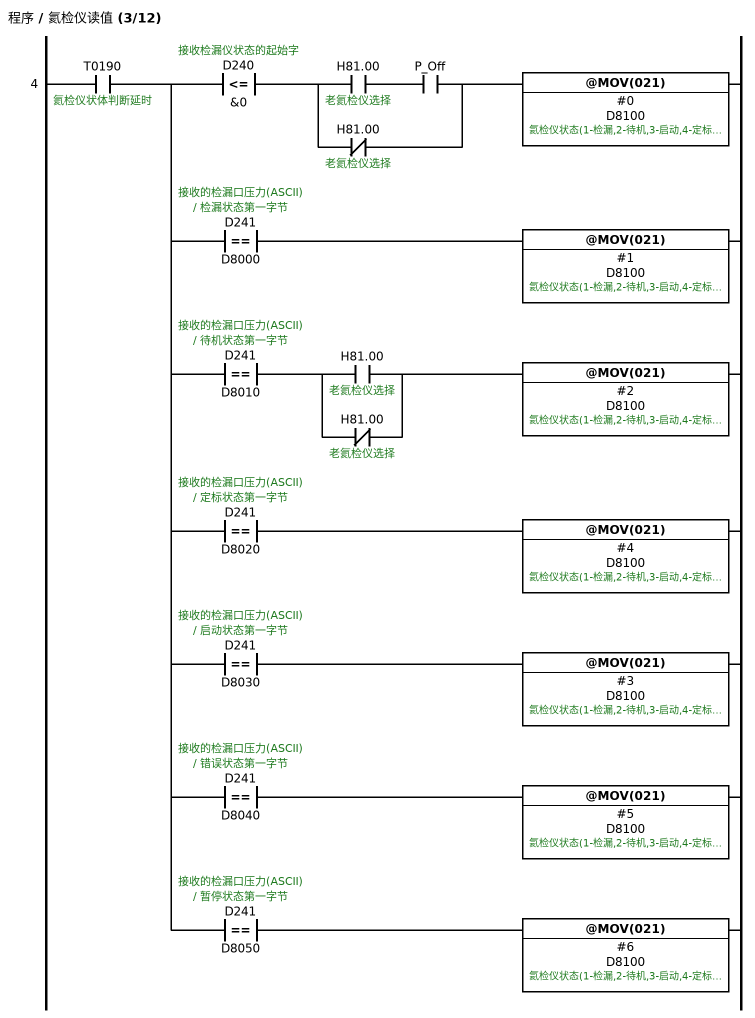
; rung 4
LD T0190  ; 氦检仪状体判断延时
OUT TR0
AND<=(315) D240 &0  ; 接收检漏仪状态的起始字
LD H81.00  ; 老氦检仪选择
AND P_Off
ORNOT H81.00  ; 老氦检仪选择
ANDLD
@MOV(021) #0 D8100  ; 氦检仪状态(1-检漏,2-待机,3-启动,4-定标,5-错误,6-暂停)
LD TR0
AND=(300) D241 D8000  ; 接收的检漏口压力(ASCII), 检漏状态第一字节
@MOV(021) #1 D8100  ; 氦检仪状态(1-检漏,2-待机,3-启动,4-定标,5-错误,6-暂停)
LD TR0
AND=(300) D241 D8010  ; 接收的检漏口压力(ASCII), 待机状态第一字节
LD H81.00  ; 老氦检仪选择
ORNOT H81.00  ; 老氦检仪选择
ANDLD
@MOV(021) #2 D8100  ; 氦检仪状态(1-检漏,2-待机,3-启动,4-定标,5-错误,6-暂停)
LD TR0
AND=(300) D241 D8020  ; 接收的检漏口压力(ASCII), 定标状态第一字节
@MOV(021) #4 D8100  ; 氦检仪状态(1-检漏,2-待机,3-启动,4-定标,5-错误,6-暂停)
LD TR0
AND=(300) D241 D8030  ; 接收的检漏口压力(ASCII), 启动状态第一字节
@MOV(021) #3 D8100  ; 氦检仪状态(1-检漏,2-待机,3-启动,4-定标,5-错误,6-暂停)
LD TR0
AND=(300) D241 D8040  ; 接收的检漏口压力(ASCII), 错误状态第一字节
@MOV(021) #5 D8100  ; 氦检仪状态(1-检漏,2-待机,3-启动,4-定标,5-错误,6-暂停)
LD TR0
AND=(300) D241 D8050  ; 接收的检漏口压力(ASCII), 暂停状态第一字节
@MOV(021) #6 D8100  ; 氦检仪状态(1-检漏,2-待机,3-启动,4-定标,5-错误,6-暂停)

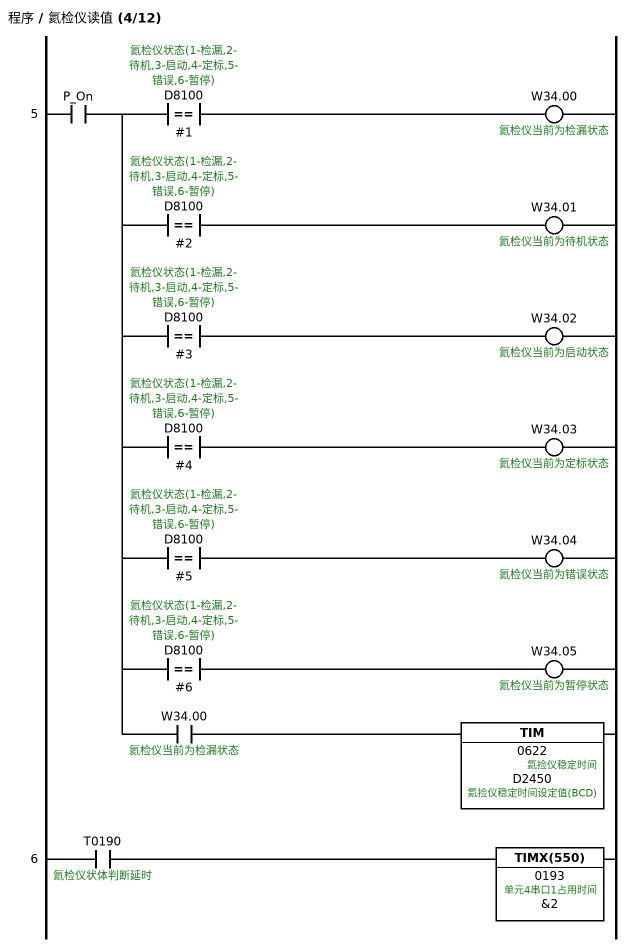
; rung 5
LD P_On
OUT TR0
AND=(300) D8100 #1  ; 氦检仪状态(1-检漏,2-待机,3-启动,4-定标,5-错误,6-暂停)
OUT W34.00  ; 氦检仪当前为检漏状态
LD TR0
AND=(300) D8100 #2  ; 氦检仪状态(1-检漏,2-待机,3-启动,4-定标,5-错误,6-暂停)
OUT W34.01  ; 氦检仪当前为待机状态
LD TR0
AND=(300) D8100 #3  ; 氦检仪状态(1-检漏,2-待机,3-启动,4-定标,5-错误,6-暂停)
OUT W34.02  ; 氦检仪当前为启动状态
LD TR0
AND=(300) D8100 #4  ; 氦检仪状态(1-检漏,2-待机,3-启动,4-定标,5-错误,6-暂停)
OUT W34.03  ; 氦检仪当前为定标状态
LD TR0
AND=(300) D8100 #5  ; 氦检仪状态(1-检漏,2-待机,3-启动,4-定标,5-错误,6-暂停)
OUT W34.04  ; 氦检仪当前为错误状态
LD TR0
AND=(300) D8100 #6  ; 氦检仪状态(1-检漏,2-待机,3-启动,4-定标,5-错误,6-暂停)
OUT W34.05  ; 氦检仪当前为暂停状态
LD TR0
AND W34.00  ; 氦检仪当前为检漏状态
TIM 0622 D2450  ; 氦捡仪稳定时间设定值(BCD), 氦捡仪稳定时间
; rung 6
LD T0190  ; 氦检仪状体判断延时
TIMX(550) 0193 &2  ; 单元4串口1占用时间

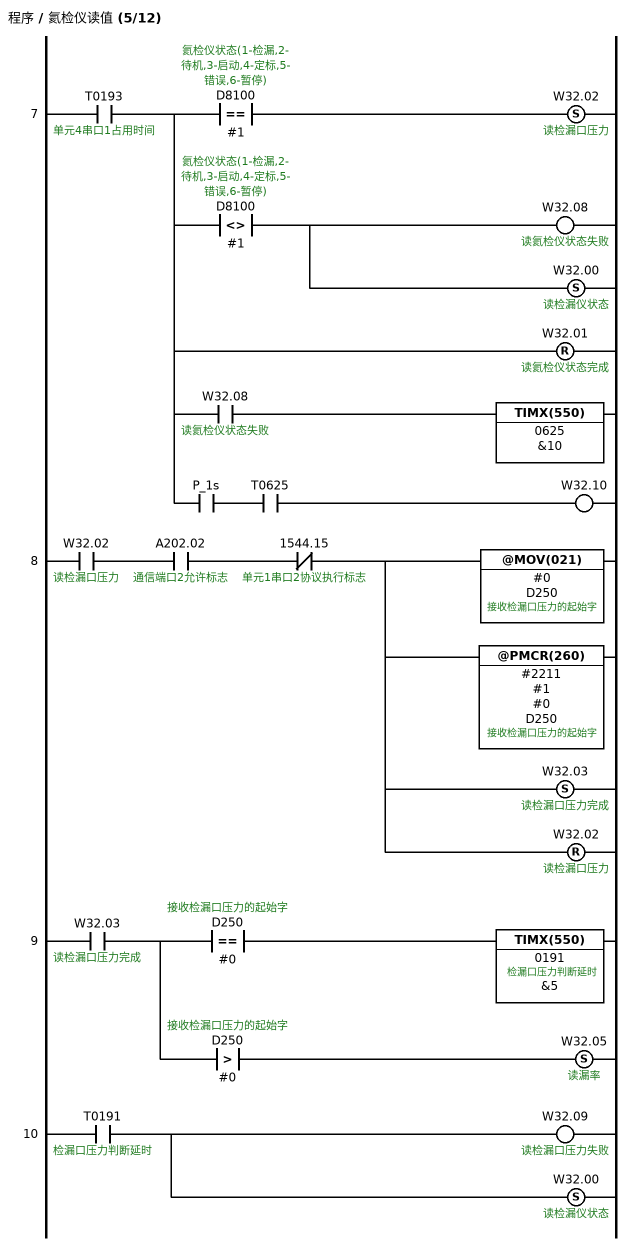
; rung 7
LD T0193  ; 单元4串口1占用时间
OUT TR0
AND=(300) D8100 #1  ; 氦检仪状态(1-检漏,2-待机,3-启动,4-定标,5-错误,6-暂停)
SET W32.02  ; 读检漏口压力
LD TR0
AND<>(305) D8100 #1  ; 氦检仪状态(1-检漏,2-待机,3-启动,4-定标,5-错误,6-暂停)
OUT W32.08  ; 读氦检仪状态失败
SET W32.00  ; 读检漏仪状态
LD TR0
RSET W32.01  ; 读氦检仪状态完成
AND W32.08  ; 读氦检仪状态失败
TIMX(550) 0625 &10
LD TR0
AND P_1s
AND T0625
OUT W32.10
; rung 8
LD W32.02  ; 读检漏口压力
AND A202.02  ; 通信端口2允许标志
ANDNOT 1544.15  ; 单元1串口2协议执行标志
@MOV(021) #0 D250  ; 接收检漏口压力的起始字
@PMCR(260) #2211 #1 #0 D250  ; 接收检漏口压力的起始字
SET W32.03  ; 读检漏口压力完成
RSET W32.02  ; 读检漏口压力
; rung 9
LD W32.03  ; 读检漏口压力完成
OUT TR0
AND=(300) D250 #0  ; 接收检漏口压力的起始字
TIMX(550) 0191 &5  ; 检漏口压力判断延时
LD TR0
AND>(320) D250 #0  ; 接收检漏口压力的起始字
SET W32.05  ; 读漏率
; rung 10
LD T0191  ; 检漏口压力判断延时
OUT W32.09  ; 读检漏口压力失败
SET W32.00  ; 读检漏仪状态

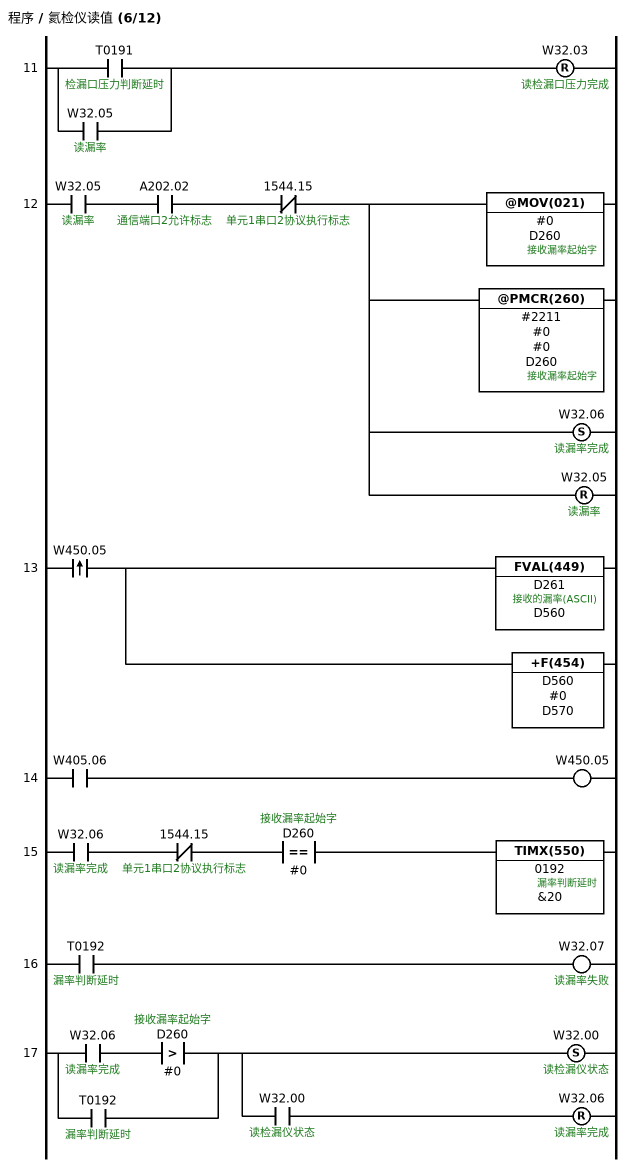
; rung 11
LD T0191  ; 检漏口压力判断延时
OR W32.05  ; 读漏率
RSET W32.03  ; 读检漏口压力完成
; rung 12
LD W32.05  ; 读漏率
AND A202.02  ; 通信端口2允许标志
ANDNOT 1544.15  ; 单元1串口2协议执行标志
@MOV(021) #0 D260  ; 接收漏率起始字
@PMCR(260) #2211 #0 #0 D260  ; 接收漏率起始字
SET W32.06  ; 读漏率完成
RSET W32.05  ; 读漏率
; rung 13
@LD W450.05
FVAL(449) D261 D560  ; 接收的漏率(ASCII)
+F(454) D560 #0 D570
; rung 14
LD W405.06
OUT W450.05
; rung 15
LD W32.06  ; 读漏率完成
ANDNOT 1544.15  ; 单元1串口2协议执行标志
AND=(300) D260 #0  ; 接收漏率起始字
TIMX(550) 0192 &20  ; 漏率判断延时
; rung 16
LD T0192  ; 漏率判断延时
OUT W32.07  ; 读漏率失败
; rung 17
LD W32.06  ; 读漏率完成
AND>(320) D260 #0  ; 接收漏率起始字
OR T0192  ; 漏率判断延时
SET W32.00  ; 读检漏仪状态
AND W32.00  ; 读检漏仪状态
RSET W32.06  ; 读漏率完成

